// TIA Portal V20 export
FUNCTION_BLOCK "Fx_LadBoxes"   // FB4, LAD
{ S7_Optimized_Access := 'TRUE' }
// stored: MemoryReserve 100, SetENOAutomatically false
   VAR_INPUT
      go : Bool;
      rst : Bool;
      n : Int;
      x : Int;
   END_VAR
   VAR_OUTPUT
      late : Bool;
      elapsed : Time;
      full : Bool;
      count : Int;
      big : Bool;
      within : Bool;
      m1 : Int;
      m2 : Int;
      sum : Int;
      "real" : Real;
      ret : Int;
      done : Bool;
   END_VAR
   VAR
      delay : TON_TIME;
   END_VAR
   VAR RETAIN
      ctr : CTU_INT;
   END_VAR
   VAR_TEMP   // added for the SCL form of the ladder/FBD networks
      _w1 : Bool;
   END_VAR
BEGIN

REGION Network 1
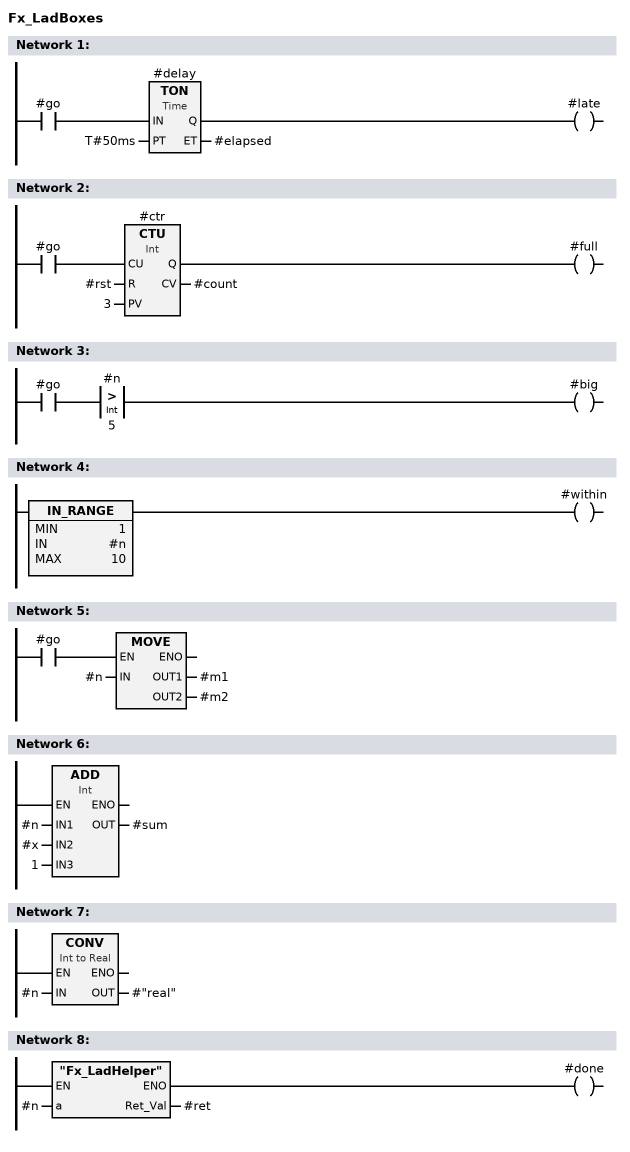
   RUNG wire#powerrail
      Contact( #go )
      { S7_Templates := "time_type := Time" } #delay.TON(pt := T#50ms, et => #elapsed)
      Coil( #late )
   END_RUNG
   // the same network as SCL:
   #delay(IN := #go, PT := T#50ms, ET => #elapsed);   // TON
   #late := #delay.Q;
END_REGION

REGION Network 2
   RUNG wire#powerrail
      Contact( #go )
      { S7_Templates := "value_type := Int" } #ctr.CTU(r := #rst, pv := 3, cv => #count)
      Coil( #full )
   END_RUNG
   // the same network as SCL:
   #ctr(CU := #go, R := #rst, PV := 3, CV => #count);   // CTU
   #full := #ctr.Q;
END_REGION

REGION Network 3
   RUNG wire#powerrail
      Contact( #go )
      { S7_Templates := "SrcType := Int" } GT_Contact(in1 := #n, in2 := 5)
      Coil( #big )
   END_RUNG
   // the same network as SCL:
   #big := #go AND (#n > 5);
END_REGION

REGION Network 4
   RUNG wire#powerrail
      { S7_Templates := "SrcType := Int" } InRange(min := 1, in := #n, max := 10)
      Coil( #within )
   END_RUNG
   // the same network as SCL:
   #within := (1 <= #n) AND (#n <= 10);
END_REGION

REGION Network 5
   RUNG wire#powerrail
      Contact( #go )
      { S7_GenerateENO := "TRUE" } Move(in := #n, out1 => #m1, out2 => #m2)
   END_RUNG
   // the same network as SCL:
   IF #go THEN
       #m1 := #n;
       #m2 := #n;
   END_IF;
END_REGION

REGION Network 6
   RUNG wire#powerrail
      { S7_Templates := "SrcType := Int"; S7_GenerateENO := "TRUE" } Add(in1 := #n, in2 := #x, in3 := 1, out => #sum)
   END_RUNG
   // the same network as SCL:
   #sum := #n + #x + 1;
END_REGION

REGION Network 7
   RUNG wire#powerrail
      { S7_Templates := "[SrcType := Int, DestType := Real]"; S7_GenerateENO := "TRUE" } Convert(in := #n, out => #"real")
   END_RUNG
   // the same network as SCL:
   #"real" := INT_TO_REAL(#n);
END_REGION

REGION Network 8
   RUNG wire#powerrail
      "Fx_LadHelper"("a" := #n, Ret_Val => #ret)
      Coil( #done )
   END_RUNG
   // the same network as SCL:
   #ret := "Fx_LadHelper"("a" := #n, ENO => #_w1);
   #done := #_w1;
END_REGION
END_FUNCTION_BLOCK
